{attribute 'linkalways'}
{attribute 'no_explicit_call' := 'do not call this POU directly'}
FUNCTION_BLOCK Dictionary
VAR
END_VAR

METHOD PUBLIC AddKeyValue
VAR_INPUT
	Key : T_MAXSTRING;
	Value : ANY;
END_VAR
END_METHOD

METHOD PUBLIC Clear
VAR_INPUT
END_VAR
END_METHOD

METHOD PUBLIC ContainsKey : BOOL;
VAR_INPUT
	Key : T_MAXSTRING;
END_VAR
END_METHOD

PROPERTY PUBLIC Count : UINT
GET
VAR
	currentCount : UINT;
	currentItem : I_DictionaryItem;
END_VAR
END_GET
END_PROPERTY

METHOD PRIVATE GetItemByKey : I_DictionaryItem
VAR_INPUT
	Key : T_MAXSTRING;
END_VAR
END_METHOD

METHOD PUBLIC Remove
VAR_INPUT
	Key : T_MAXSTRING;
END_VAR
END_METHOD

METHOD PUBLIC TryGetValue : BOOL;
VAR_INPUT
	Key : T_MAXSTRING;
	Destination : ANY;
END_VAR
END_METHOD

END_FUNCTION_BLOCK

(* stored: Version 1.1.0.1, ProductVersion 3.1.4024.12
   POU Dictionary: Id {2496496f-6f27-4201-9f0e-92026c6200d3}, SpecialFunc None
   Folder Private: Id {d1bfc11a-bfb8-4279-8f99-8ed64ee1dde6}
   Method AddKeyValue: Id {d65f77f4-4ccd-40df-9fd0-75019b8c0eda}
   Method Clear: Id {7785c898-3c48-4fe2-81e1-cacbbc4b08af}
   Method ContainsKey: Id {c30a7e26-67f2-4551-b9c7-e531d1461757}
   Property Count: Id {9ebe98eb-1d50-4553-a45d-3da249d13a8f}
   Get Get: Id {1c0d3937-4ab9-4f4e-aaa8-c17c25b4cf78}
   Method GetItemByKey: Id {af2545c1-cc5f-4ca6-921c-5788cb2a81eb}
   Method Remove: Id {a24dcb40-efa1-4f1e-a731-a3646f2b28cd}
   Method TryGetValue: Id {e9df9db0-5f25-404e-929c-5a02ea131685} *)
